(* Logix 5000 project; controller configured_IO_modules vendor 1 type 14 code 106 rev 28.11; software revision 28.03 *)

TASK MainTask (continuous, watchdog 500 ms) : MainProgram

MODULES
   Local : vendor 1 type 14 code 106 (Compact 0, rev 28.11)
       : vendor 1 type 7 code 77 (Compact 2, rev 3.1, Input RPI 20 ms)
       : 1769-IQ16 (Compact 3, rev 1.1, Input RPI 20 ms)
       : vendor 1 type 7 code 72 (Compact 5, rev 2.1, Output RPI 20 ms)
       : vendor 1 type 7 code 72 (Compact 4, rev 2.1, Output RPI 20 ms)
END_MODULES

PROGRAM MainProgram   (* main routine MainRoutine *)

ROUTINE MainRoutine   (* ladder *)
END_ROUTINE
END_PROGRAM
